TYPE STATE:
    STRUCT
        curTime: LREAL;
        dvar_M_p_b AT %Q*: BOOL;
        dvar_M_p_x AT %Q*: DINT;
        dvar_M_p_y AT %Q*: LREAL;
        dvar_M_p_ve AT %Q*: enum_E;
        dvar_M_p_v1 AT %Q*: DINT;
        dvar_M_p_v2 AT %Q*: TupleStruct_1;
        dvar_M_p_v3 AT %Q*: TupleStruct_2;
        dvar_M_p_tv AT %Q*: TupleStruct_3;
        dvar_M_p_j AT %Q*: DINT;
        dvar_M_p_r AT %Q*: LREAL;
        cvar_M_p_t AT %Q*: LREAL;
        cvar_M_p_t2 AT %Q*: LREAL;
        cvar_M_p_t3 AT %Q*: LREAL;
        dvar_M_p AT %Q*: enum_E;
    END_STRUCT
END_TYPE

(* stored: ProductVersion 3.1.0.18, Version 1.1.0.1 *)
